VAR_GLOBAL
	FaultCheck_G : BOOL ; // Test if Fault 
	Fault_Count_G: CTU  ; // Counter 	
	

END_VAR

(* stored: Version 1.1.0.1, ProductVersion 3.1.4024.6
   GVL GVL_Check: Id {f5694ae6-cd0e-420d-949a-4d1e24e09fad} *)
